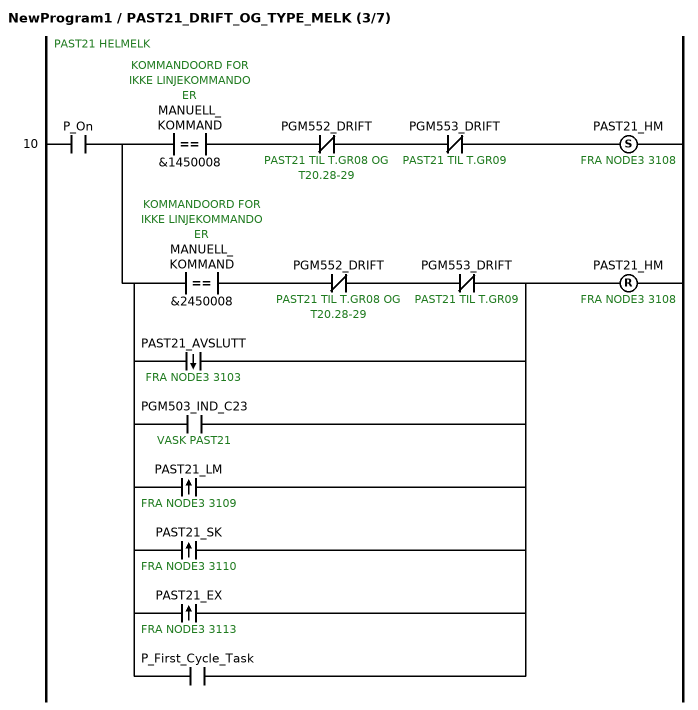
; [picture p1032: NewProgram1 / PAST21_DRIFT_OG_TYPE_MELK, rungs 10-10]
; rung 10: PAST21 HELMELK
LD P_On
OUT TR0
AND=L(301) MANUELL_KOMMAND &1450008  ; KOMMANDOORD FOR IKKE LINJEKOMMANDOER
ANDNOT PGM552_DRIFT  ; PAST21 TIL T.GR08 OG T20.28-29
ANDNOT PGM553_DRIFT  ; PAST21 TIL T.GR09
SET PAST21_HM  ; FRA NODE3 3108
LD TR0
LD=L(301) MANUELL_KOMMAND &2450008  ; KOMMANDOORD FOR IKKE LINJEKOMMANDOER
ANDNOT PGM552_DRIFT  ; PAST21 TIL T.GR08 OG T20.28-29
ANDNOT PGM553_DRIFT  ; PAST21 TIL T.GR09
%OR PAST21_AVSLUTT  ; FRA NODE3 3103
OR PGM503_IND_C23  ; VASK PAST21
@OR PAST21_LM  ; FRA NODE3 3109
@OR PAST21_SK  ; FRA NODE3 3110
@OR PAST21_EX  ; FRA NODE3 3113
OR P_First_Cycle_Task
ANDLD
RSET PAST21_HM  ; FRA NODE3 3108

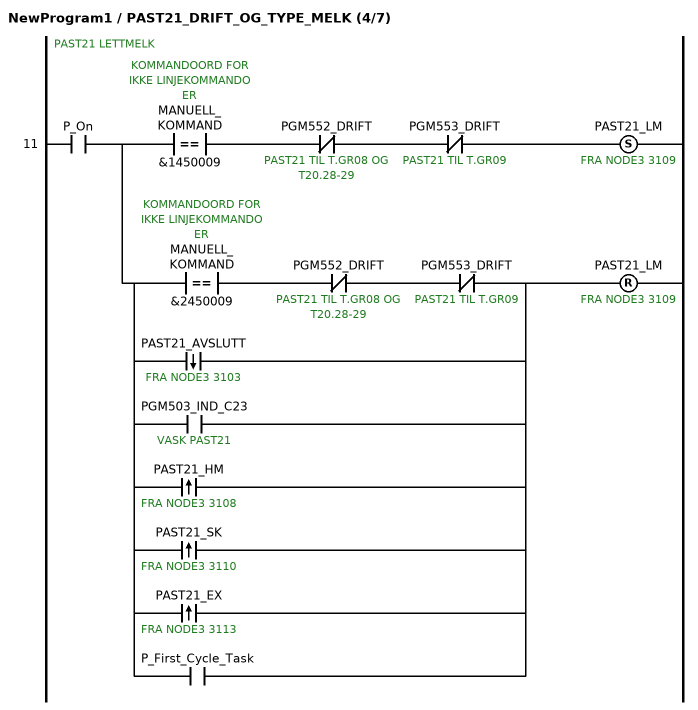
; rung 11: PAST21 LETTMELK
LD P_On
OUT TR0
AND=L(301) MANUELL_KOMMAND &1450009  ; KOMMANDOORD FOR IKKE LINJEKOMMANDOER
ANDNOT PGM552_DRIFT  ; PAST21 TIL T.GR08 OG T20.28-29
ANDNOT PGM553_DRIFT  ; PAST21 TIL T.GR09
SET PAST21_LM  ; FRA NODE3 3109
LD TR0
LD=L(301) MANUELL_KOMMAND &2450009  ; KOMMANDOORD FOR IKKE LINJEKOMMANDOER
ANDNOT PGM552_DRIFT  ; PAST21 TIL T.GR08 OG T20.28-29
ANDNOT PGM553_DRIFT  ; PAST21 TIL T.GR09
%OR PAST21_AVSLUTT  ; FRA NODE3 3103
OR PGM503_IND_C23  ; VASK PAST21
@OR PAST21_HM  ; FRA NODE3 3108
@OR PAST21_SK  ; FRA NODE3 3110
@OR PAST21_EX  ; FRA NODE3 3113
OR P_First_Cycle_Task
ANDLD
RSET PAST21_LM  ; FRA NODE3 3109

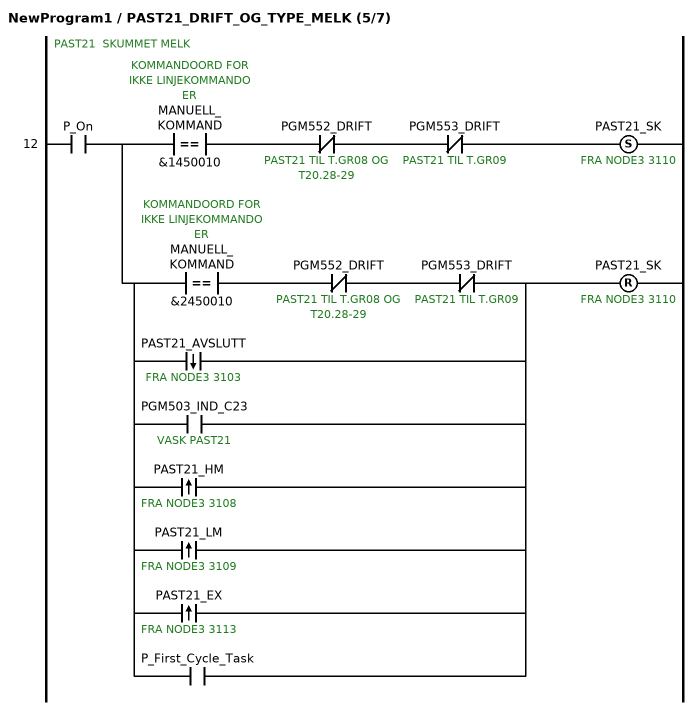
; rung 12: PAST21  SKUMMET MELK
LD P_On
OUT TR0
AND=L(301) MANUELL_KOMMAND &1450010  ; KOMMANDOORD FOR IKKE LINJEKOMMANDOER
ANDNOT PGM552_DRIFT  ; PAST21 TIL T.GR08 OG T20.28-29
ANDNOT PGM553_DRIFT  ; PAST21 TIL T.GR09
SET PAST21_SK  ; FRA NODE3 3110
LD TR0
LD=L(301) MANUELL_KOMMAND &2450010  ; KOMMANDOORD FOR IKKE LINJEKOMMANDOER
ANDNOT PGM552_DRIFT  ; PAST21 TIL T.GR08 OG T20.28-29
ANDNOT PGM553_DRIFT  ; PAST21 TIL T.GR09
%OR PAST21_AVSLUTT  ; FRA NODE3 3103
OR PGM503_IND_C23  ; VASK PAST21
@OR PAST21_HM  ; FRA NODE3 3108
@OR PAST21_LM  ; FRA NODE3 3109
@OR PAST21_EX  ; FRA NODE3 3113
OR P_First_Cycle_Task
ANDLD
RSET PAST21_SK  ; FRA NODE3 3110

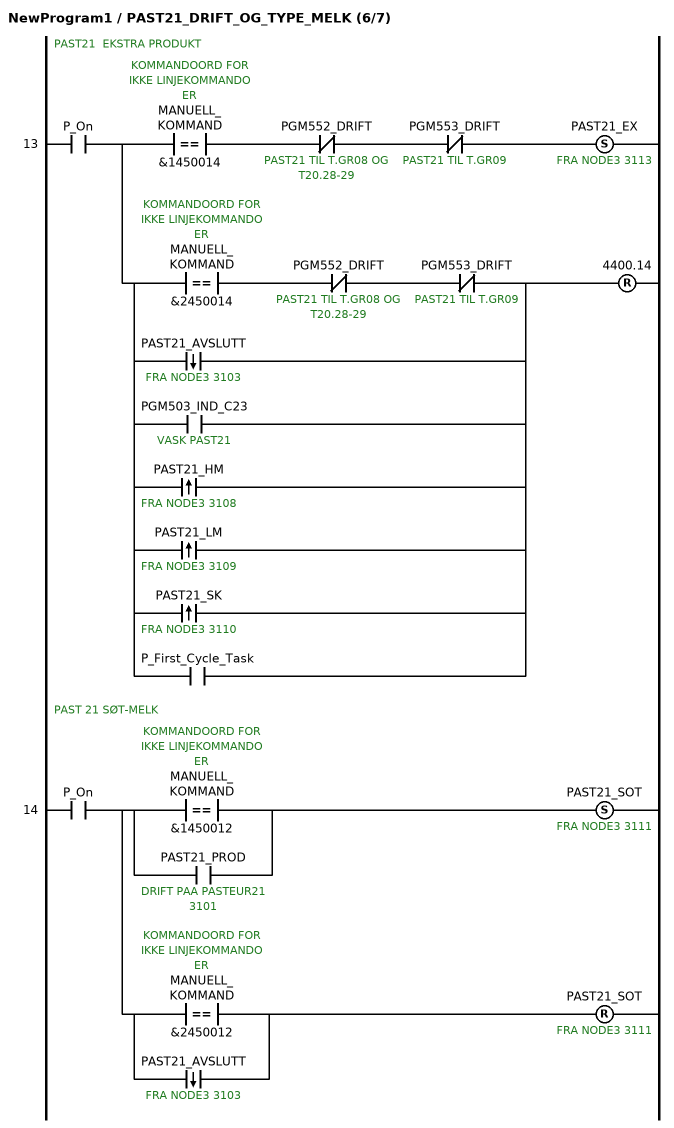
; rung 13: PAST21  EKSTRA PRODUKT
LD P_On
OUT TR0
AND=L(301) MANUELL_KOMMAND &1450014  ; KOMMANDOORD FOR IKKE LINJEKOMMANDOER
ANDNOT PGM552_DRIFT  ; PAST21 TIL T.GR08 OG T20.28-29
ANDNOT PGM553_DRIFT  ; PAST21 TIL T.GR09
SET PAST21_EX  ; FRA NODE3 3113
LD TR0
LD=L(301) MANUELL_KOMMAND &2450014  ; KOMMANDOORD FOR IKKE LINJEKOMMANDOER
ANDNOT PGM552_DRIFT  ; PAST21 TIL T.GR08 OG T20.28-29
ANDNOT PGM553_DRIFT  ; PAST21 TIL T.GR09
%OR PAST21_AVSLUTT  ; FRA NODE3 3103
OR PGM503_IND_C23  ; VASK PAST21
@OR PAST21_HM  ; FRA NODE3 3108
@OR PAST21_LM  ; FRA NODE3 3109
@OR PAST21_SK  ; FRA NODE3 3110
OR P_First_Cycle_Task
ANDLD
RSET 4400.14
; rung 14: PAST 21 SØT-MELK
LD P_On
OUT TR0
LD=L(301) MANUELL_KOMMAND &1450012  ; KOMMANDOORD FOR IKKE LINJEKOMMANDOER
OR PAST21_PROD  ; DRIFT PAA PASTEUR21 3101
ANDLD
SET PAST21_SOT  ; FRA NODE3 3111
LD TR0
LD=L(301) MANUELL_KOMMAND &2450012  ; KOMMANDOORD FOR IKKE LINJEKOMMANDOER
%OR PAST21_AVSLUTT  ; FRA NODE3 3103
ANDLD
RSET PAST21_SOT  ; FRA NODE3 3111

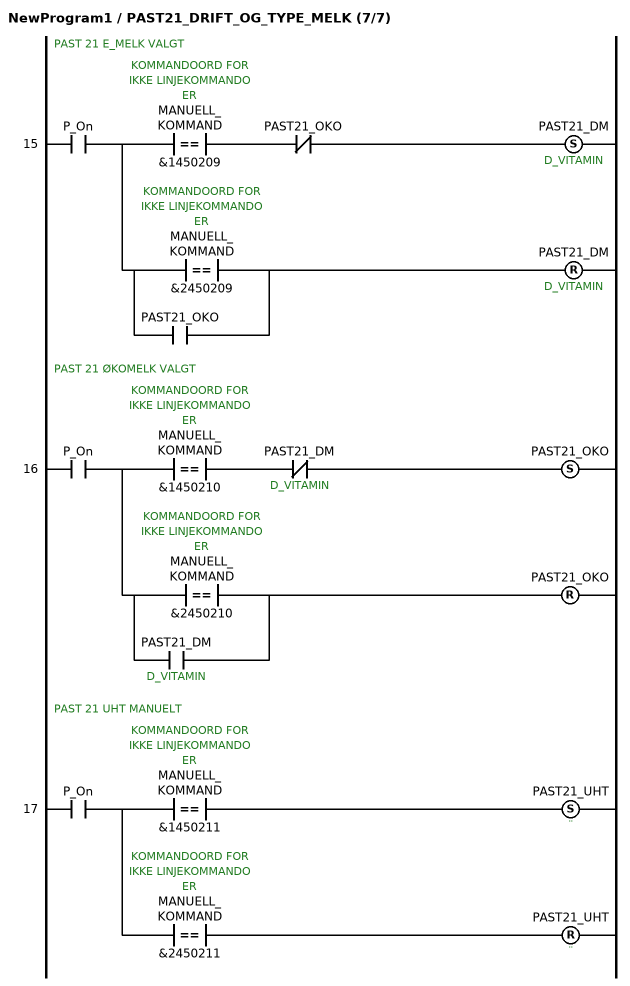
; rung 15: PAST 21 E_MELK VALGT
LD P_On
OUT TR0
AND=L(301) MANUELL_KOMMAND &1450209  ; KOMMANDOORD FOR IKKE LINJEKOMMANDOER
ANDNOT PAST21_OKO
SET PAST21_DM  ; D_VITAMIN
LD TR0
LD=L(301) MANUELL_KOMMAND &2450209  ; KOMMANDOORD FOR IKKE LINJEKOMMANDOER
OR PAST21_OKO
ANDLD
RSET PAST21_DM  ; D_VITAMIN
; rung 16: PAST 21 ØKOMELK VALGT
LD P_On
OUT TR0
AND=L(301) MANUELL_KOMMAND &1450210  ; KOMMANDOORD FOR IKKE LINJEKOMMANDOER
ANDNOT PAST21_DM  ; D_VITAMIN
SET PAST21_OKO
LD TR0
LD=L(301) MANUELL_KOMMAND &2450210  ; KOMMANDOORD FOR IKKE LINJEKOMMANDOER
OR PAST21_DM  ; D_VITAMIN
ANDLD
RSET PAST21_OKO
; rung 17: PAST 21 UHT MANUELT
LD P_On
OUT TR0
AND=L(301) MANUELL_KOMMAND &1450211  ; KOMMANDOORD FOR IKKE LINJEKOMMANDOER
SET PAST21_UHT  ; ¨
LD TR0
AND=L(301) MANUELL_KOMMAND &2450211  ; KOMMANDOORD FOR IKKE LINJEKOMMANDOER
RSET PAST21_UHT  ; ¨
; rung 18: Ingen_kommentar_funnet

### Section PAST21_STATUSKONTROLL

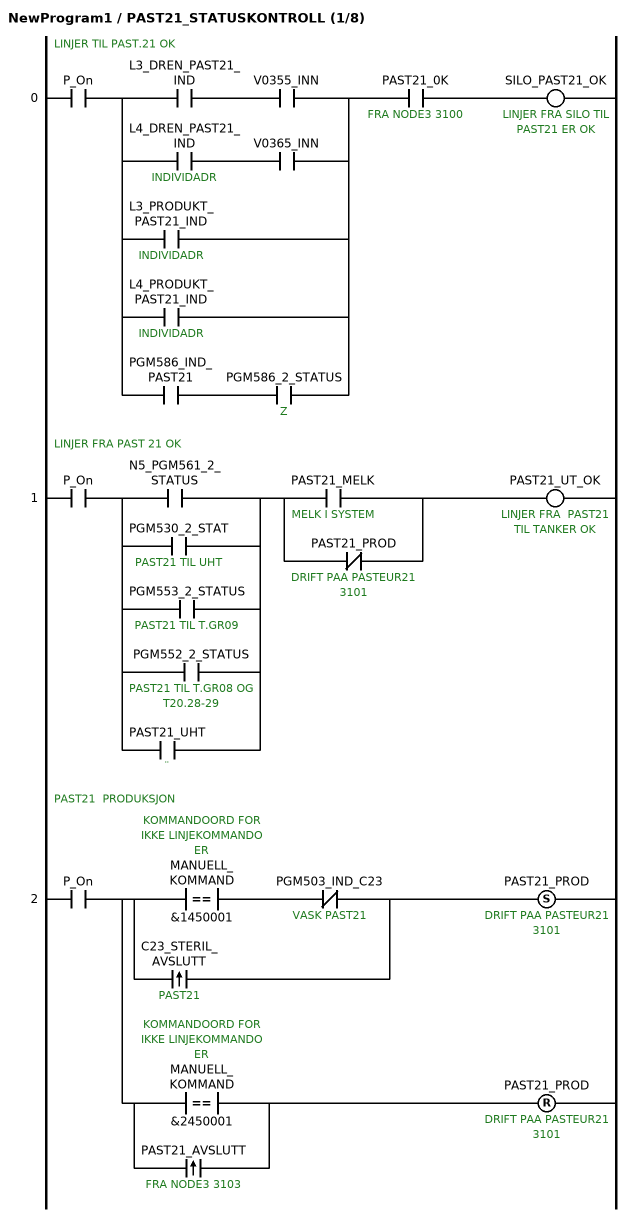
; rung 0: LINJER TIL PAST.21 OK
LD P_On
LD L3_DREN_PAST21_IND
AND V0355_INN
LD L4_DREN_PAST21_IND  ; INDIVIDADR
AND V0365_INN
ORLD
OR L3_PRODUKT_PAST21_IND  ; INDIVIDADR
OR L4_PRODUKT_PAST21_IND  ; INDIVIDADR
LD PGM586_IND_PAST21
AND PGM586_2_STATUS  ; Z
ORLD
ANDLD
AND PAST21_0K  ; FRA NODE3 3100
OUT SILO_PAST21_OK  ; LINJER FRA SILO TIL  PAST21 ER OK
; rung 1: LINJER FRA PAST 21 OK
LD P_On
LD N5_PGM561_2_STATUS
OR PGM530_2_STAT  ; PAST21 TIL UHT
OR PGM553_2_STATUS  ; PAST21 TIL T.GR09
OR PGM552_2_STATUS  ; PAST21 TIL T.GR08 OG T20.28-29
OR PAST21_UHT  ; ¨
ANDLD
LD PAST21_MELK  ; MELK I SYSTEM
ORNOT PAST21_PROD  ; DRIFT PAA PASTEUR21 3101
ANDLD
OUT PAST21_UT_OK  ; LINJER FRA  PAST21 TIL TANKER OK
; rung 2: PAST21  PRODUKSJON
LD P_On
OUT TR0
LD=L(301) MANUELL_KOMMAND &1450001  ; KOMMANDOORD FOR IKKE LINJEKOMMANDOER
ANDNOT PGM503_IND_C23  ; VASK PAST21
@OR C23_STERIL_AVSLUTT  ; PAST21
ANDLD
SET PAST21_PROD  ; DRIFT PAA PASTEUR21 3101
LD TR0
LD=L(301) MANUELL_KOMMAND &2450001  ; KOMMANDOORD FOR IKKE LINJEKOMMANDOER
@OR PAST21_AVSLUTT  ; FRA NODE3 3103
ANDLD
RSET PAST21_PROD  ; DRIFT PAA PASTEUR21 3101

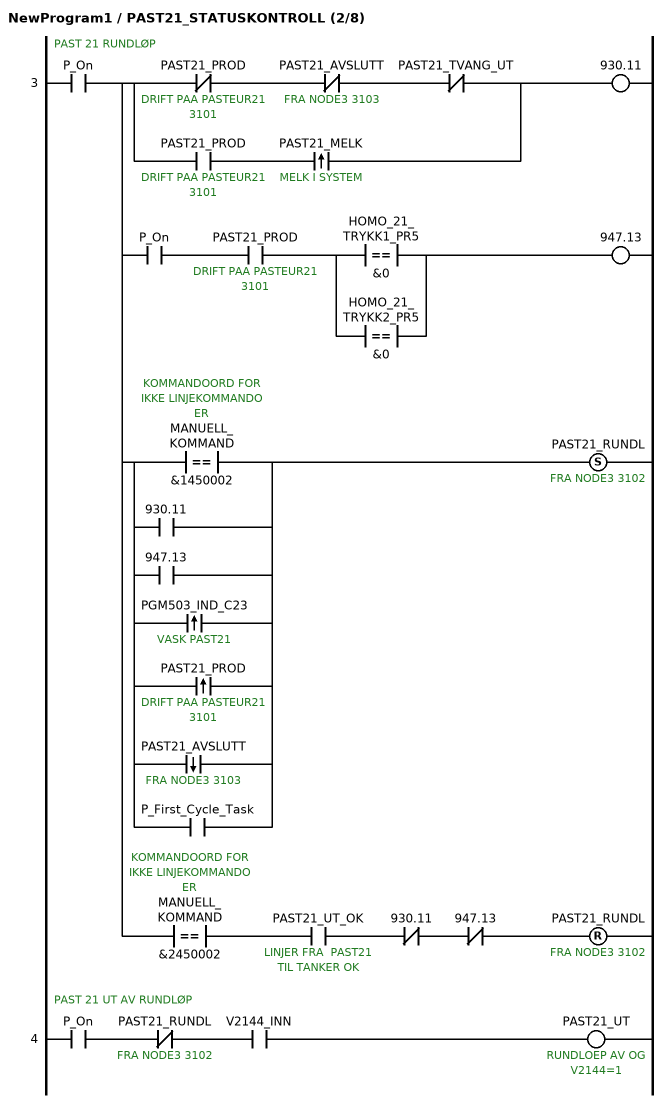
; rung 3: PAST 21 RUNDLØP
LD P_On
OUT TR0
LDNOT PAST21_PROD  ; DRIFT PAA PASTEUR21 3101
ANDNOT PAST21_AVSLUTT  ; FRA NODE3 3103
ANDNOT PAST21_TVANG_UT
LD PAST21_PROD  ; DRIFT PAA PASTEUR21 3101
@AND PAST21_MELK  ; MELK I SYSTEM
ORLD
ANDLD
OUT 930.11
LD TR0
AND P_On
AND PAST21_PROD  ; DRIFT PAA PASTEUR21 3101
LD=L(301) HOMO_21_TRYKK1_PR5 &0
OR=L(301) HOMO_21_TRYKK2_PR5 &0
ANDLD
OUT 947.13
LD TR0
LD=L(301) MANUELL_KOMMAND &1450002  ; KOMMANDOORD FOR IKKE LINJEKOMMANDOER
OR 930.11
OR 947.13
@OR PGM503_IND_C23  ; VASK PAST21
@OR PAST21_PROD  ; DRIFT PAA PASTEUR21 3101
%OR PAST21_AVSLUTT  ; FRA NODE3 3103
OR P_First_Cycle_Task
ANDLD
SET PAST21_RUNDL  ; FRA NODE3 3102
LD TR0
AND=L(301) MANUELL_KOMMAND &2450002  ; KOMMANDOORD FOR IKKE LINJEKOMMANDOER
AND PAST21_UT_OK  ; LINJER FRA  PAST21 TIL TANKER OK
ANDNOT 930.11
ANDNOT 947.13
RSET PAST21_RUNDL  ; FRA NODE3 3102
; rung 4: PAST 21 UT AV RUNDLØP
LD P_On
ANDNOT PAST21_RUNDL  ; FRA NODE3 3102
AND V2144_INN
OUT PAST21_UT  ; RUNDLOEP AV OG V2144=1

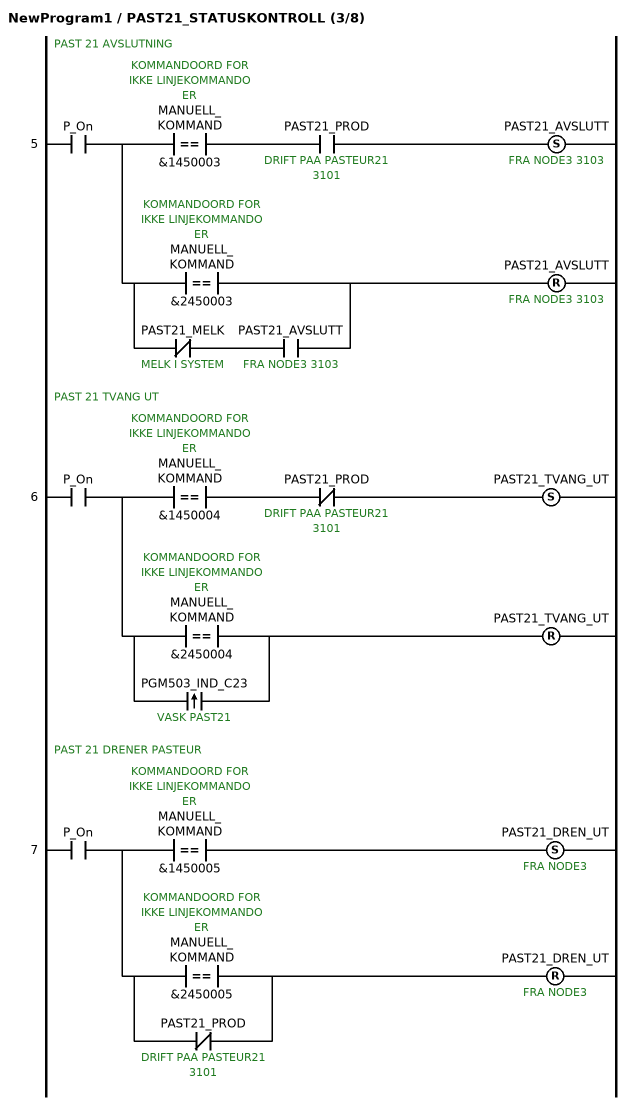
; rung 5: PAST 21 AVSLUTNING
LD P_On
OUT TR0
AND=L(301) MANUELL_KOMMAND &1450003  ; KOMMANDOORD FOR IKKE LINJEKOMMANDOER
AND PAST21_PROD  ; DRIFT PAA PASTEUR21 3101
SET PAST21_AVSLUTT  ; FRA NODE3 3103
LD TR0
LD=L(301) MANUELL_KOMMAND &2450003  ; KOMMANDOORD FOR IKKE LINJEKOMMANDOER
LDNOT PAST21_MELK  ; MELK I SYSTEM
AND PAST21_AVSLUTT  ; FRA NODE3 3103
ORLD
ANDLD
RSET PAST21_AVSLUTT  ; FRA NODE3 3103
; rung 6: PAST 21 TVANG UT
LD P_On
OUT TR0
AND=L(301) MANUELL_KOMMAND &1450004  ; KOMMANDOORD FOR IKKE LINJEKOMMANDOER
ANDNOT PAST21_PROD  ; DRIFT PAA PASTEUR21 3101
SET PAST21_TVANG_UT
LD TR0
LD=L(301) MANUELL_KOMMAND &2450004  ; KOMMANDOORD FOR IKKE LINJEKOMMANDOER
@OR PGM503_IND_C23  ; VASK PAST21
ANDLD
RSET PAST21_TVANG_UT
; rung 7: PAST 21 DRENER PASTEUR
LD P_On
OUT TR0
AND=L(301) MANUELL_KOMMAND &1450005  ; KOMMANDOORD FOR IKKE LINJEKOMMANDOER
SET PAST21_DREN_UT  ; FRA NODE3
LD TR0
LD=L(301) MANUELL_KOMMAND &2450005  ; KOMMANDOORD FOR IKKE LINJEKOMMANDOER
ORNOT PAST21_PROD  ; DRIFT PAA PASTEUR21 3101
ANDLD
RSET PAST21_DREN_UT  ; FRA NODE3

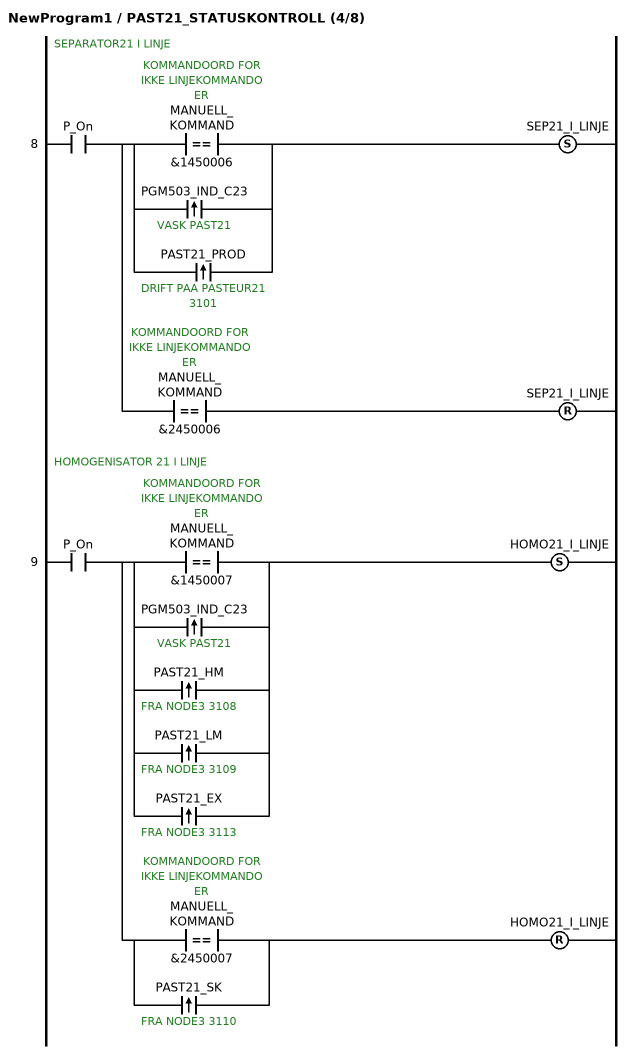
; rung 8: SEPARATOR21 I LINJE
LD P_On
OUT TR0
LD=L(301) MANUELL_KOMMAND &1450006  ; KOMMANDOORD FOR IKKE LINJEKOMMANDOER
@OR PGM503_IND_C23  ; VASK PAST21
@OR PAST21_PROD  ; DRIFT PAA PASTEUR21 3101
ANDLD
SET SEP21_I_LINJE
LD TR0
AND=L(301) MANUELL_KOMMAND &2450006  ; KOMMANDOORD FOR IKKE LINJEKOMMANDOER
RSET SEP21_I_LINJE
; rung 9: HOMOGENISATOR 21 I LINJE
LD P_On
OUT TR0
LD=L(301) MANUELL_KOMMAND &1450007  ; KOMMANDOORD FOR IKKE LINJEKOMMANDOER
@OR PGM503_IND_C23  ; VASK PAST21
@OR PAST21_HM  ; FRA NODE3 3108
@OR PAST21_LM  ; FRA NODE3 3109
@OR PAST21_EX  ; FRA NODE3 3113
ANDLD
SET HOMO21_I_LINJE
LD TR0
LD=L(301) MANUELL_KOMMAND &2450007  ; KOMMANDOORD FOR IKKE LINJEKOMMANDOER
@OR PAST21_SK  ; FRA NODE3 3110
ANDLD
RSET HOMO21_I_LINJE

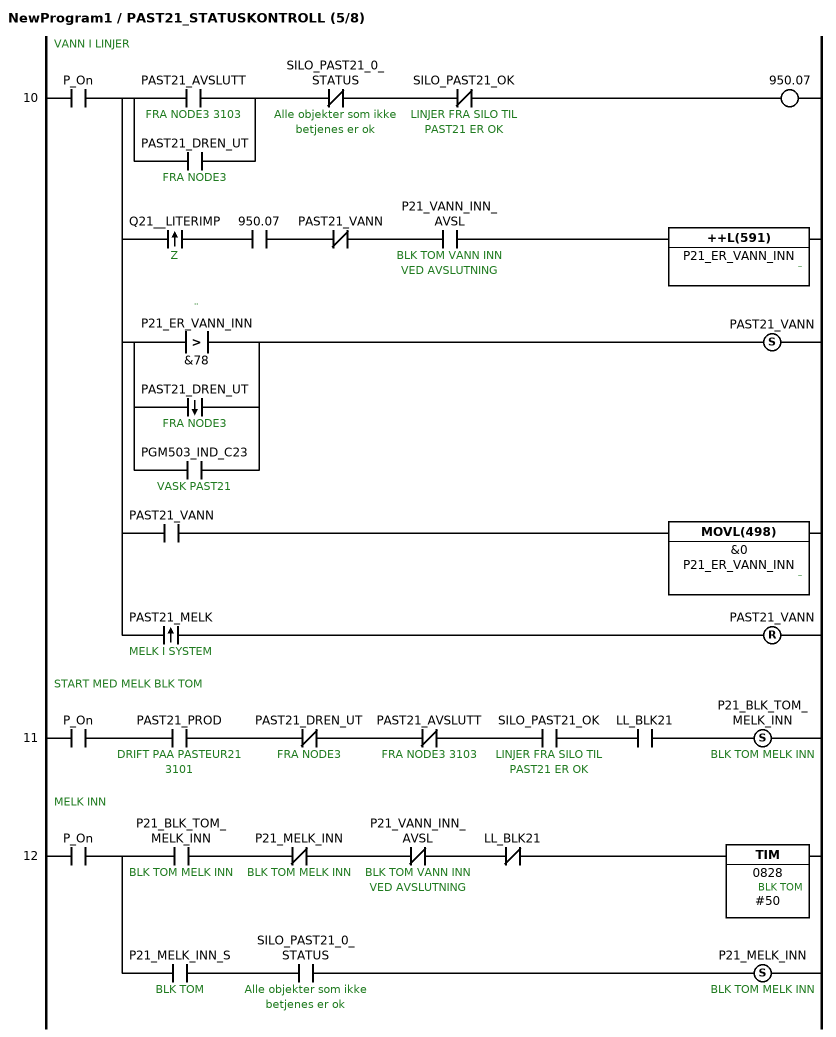
; rung 10: VANN I LINJER
LD P_On
OUT TR0
LD PAST21_AVSLUTT  ; FRA NODE3 3103
OR PAST21_DREN_UT  ; FRA NODE3
ANDLD
ANDNOT SILO_PAST21_0_STATUS  ; Alle objekter som ikke betjenes er ok
ANDNOT SILO_PAST21_OK  ; LINJER FRA SILO TIL  PAST21 ER OK
OUT 950.07
LD TR0
@AND Q21__LITERIMP  ; Z
AND 950.07
ANDNOT PAST21_VANN
AND P21_VANN_INN_AVSL  ; BLK TOM VANN INN VED AVSLUTNING
++L(591) P21_ER_VANN_INN  ; ¨
LD TR0
LD>L(321) P21_ER_VANN_INN &78  ; ¨
%OR PAST21_DREN_UT  ; FRA NODE3
OR PGM503_IND_C23  ; VASK PAST21
ANDLD
SET PAST21_VANN
LD TR0
AND PAST21_VANN
MOVL(498) &0 P21_ER_VANN_INN  ; ¨
LD TR0
@AND PAST21_MELK  ; MELK I SYSTEM
RSET PAST21_VANN
; rung 11: START MED MELK BLK TOM
LD P_On
AND PAST21_PROD  ; DRIFT PAA PASTEUR21 3101
ANDNOT PAST21_DREN_UT  ; FRA NODE3
ANDNOT PAST21_AVSLUTT  ; FRA NODE3 3103
AND SILO_PAST21_OK  ; LINJER FRA SILO TIL  PAST21 ER OK
AND LL_BLK21
SET P21_BLK_TOM_MELK_INN  ; BLK TOM MELK INN
; rung 12: MELK INN
LD P_On
OUT TR0
AND P21_BLK_TOM_MELK_INN  ; BLK TOM MELK INN
ANDNOT P21_MELK_INN  ; BLK TOM MELK INN
ANDNOT P21_VANN_INN_AVSL  ; BLK TOM VANN INN VED AVSLUTNING
ANDNOT LL_BLK21
TIM 0828 #50  ; BLK TOM
LD TR0
AND P21_MELK_INN_S  ; BLK TOM
AND SILO_PAST21_0_STATUS  ; Alle objekter som ikke betjenes er ok
SET P21_MELK_INN  ; BLK TOM MELK INN

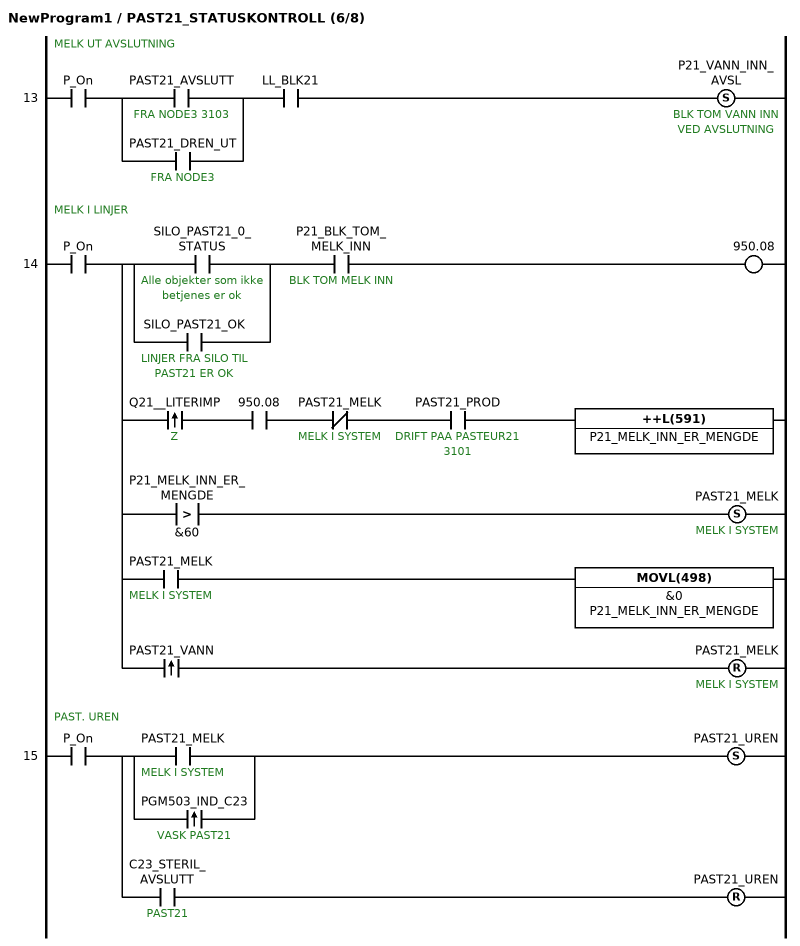
; rung 13: MELK UT AVSLUTNING
LD P_On
LD PAST21_AVSLUTT  ; FRA NODE3 3103
OR PAST21_DREN_UT  ; FRA NODE3
ANDLD
AND LL_BLK21
SET P21_VANN_INN_AVSL  ; BLK TOM VANN INN VED AVSLUTNING
; rung 14: MELK I LINJER
LD P_On
OUT TR0
LD SILO_PAST21_0_STATUS  ; Alle objekter som ikke betjenes er ok
OR SILO_PAST21_OK  ; LINJER FRA SILO TIL  PAST21 ER OK
ANDLD
AND P21_BLK_TOM_MELK_INN  ; BLK TOM MELK INN
OUT 950.08
LD TR0
@AND Q21__LITERIMP  ; Z
AND 950.08
ANDNOT PAST21_MELK  ; MELK I SYSTEM
AND PAST21_PROD  ; DRIFT PAA PASTEUR21 3101
++L(591) P21_MELK_INN_ER_MENGDE
LD TR0
AND>L(321) P21_MELK_INN_ER_MENGDE &60
SET PAST21_MELK  ; MELK I SYSTEM
LD TR0
AND PAST21_MELK  ; MELK I SYSTEM
MOVL(498) &0 P21_MELK_INN_ER_MENGDE
LD TR0
@AND PAST21_VANN
RSET PAST21_MELK  ; MELK I SYSTEM
; rung 15: PAST. UREN
LD P_On
OUT TR0
LD PAST21_MELK  ; MELK I SYSTEM
@OR PGM503_IND_C23  ; VASK PAST21
ANDLD
SET PAST21_UREN
LD TR0
AND C23_STERIL_AVSLUTT  ; PAST21
RSET PAST21_UREN

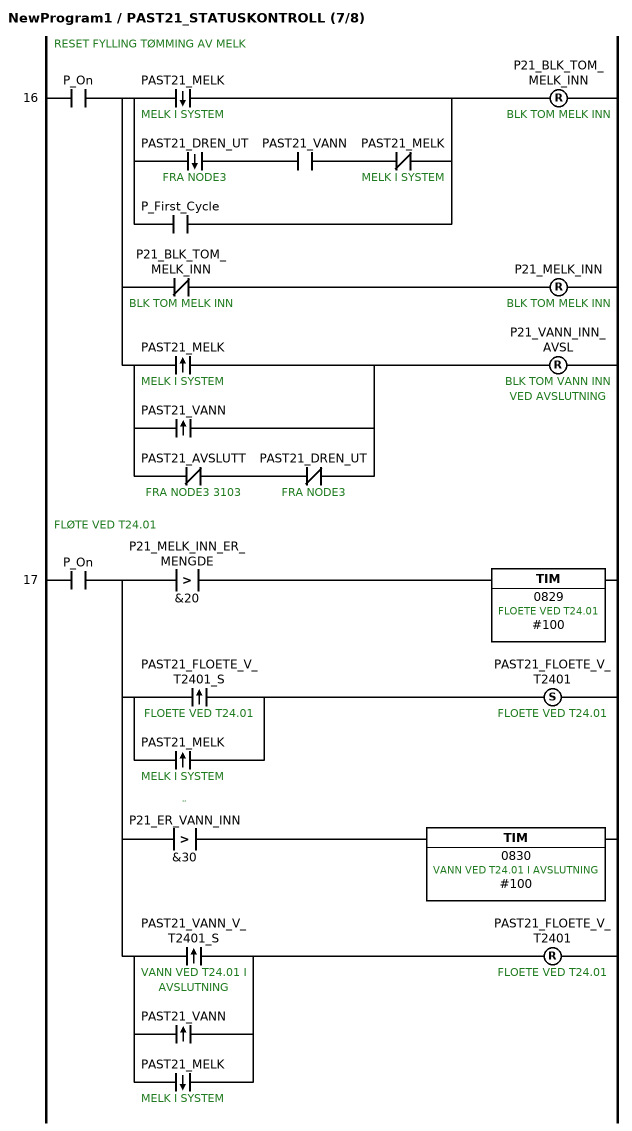
; rung 16: RESET FYLLING TØMMING AV MELK
LD P_On
OUT TR0
%LD PAST21_MELK  ; MELK I SYSTEM
%LD PAST21_DREN_UT  ; FRA NODE3
AND PAST21_VANN
ANDNOT PAST21_MELK  ; MELK I SYSTEM
ORLD
OR P_First_Cycle
ANDLD
RSET P21_BLK_TOM_MELK_INN  ; BLK TOM MELK INN
LD TR0
ANDNOT P21_BLK_TOM_MELK_INN  ; BLK TOM MELK INN
RSET P21_MELK_INN  ; BLK TOM MELK INN
LD TR0
@LD PAST21_MELK  ; MELK I SYSTEM
@OR PAST21_VANN
LDNOT PAST21_AVSLUTT  ; FRA NODE3 3103
ANDNOT PAST21_DREN_UT  ; FRA NODE3
ORLD
ANDLD
RSET P21_VANN_INN_AVSL  ; BLK TOM VANN INN VED AVSLUTNING
; rung 17: FLØTE VED T24.01
LD P_On
OUT TR0
AND>L(321) P21_MELK_INN_ER_MENGDE &20
TIM 0829 #100  ; FLOETE VED T24.01
LD TR0
@LD PAST21_FLOETE_V_T2401_S  ; FLOETE VED T24.01
@OR PAST21_MELK  ; MELK I SYSTEM
ANDLD
SET PAST21_FLOETE_V_T2401  ; FLOETE VED T24.01
LD TR0
AND>L(321) P21_ER_VANN_INN &30  ; ¨
TIM 0830 #100  ; VANN VED T24.01 I AVSLUTNING
LD TR0
@LD PAST21_VANN_V_T2401_S  ; VANN VED T24.01 I AVSLUTNING
@OR PAST21_VANN
%OR PAST21_MELK  ; MELK I SYSTEM
ANDLD
RSET PAST21_FLOETE_V_T2401  ; FLOETE VED T24.01

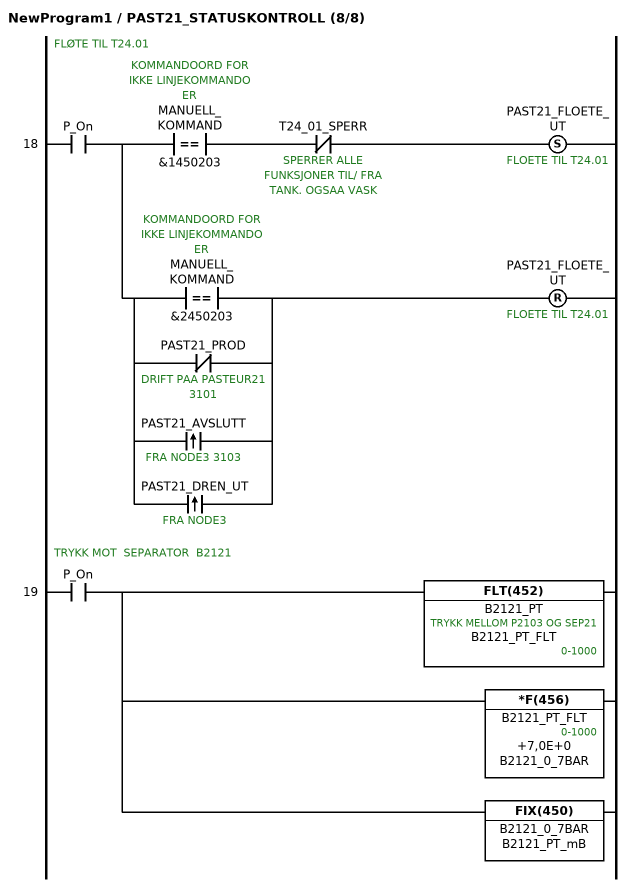
; rung 18: FLØTE TIL T24.01
LD P_On
OUT TR0
AND=L(301) MANUELL_KOMMAND &1450203  ; KOMMANDOORD FOR IKKE LINJEKOMMANDOER
ANDNOT T24_01_SPERR  ; SPERRER ALLE FUNKSJONER TIL/ FRA TANK. OGSAA VASK
SET PAST21_FLOETE_UT  ; FLOETE TIL T24.01
LD TR0
LD=L(301) MANUELL_KOMMAND &2450203  ; KOMMANDOORD FOR IKKE LINJEKOMMANDOER
ORNOT PAST21_PROD  ; DRIFT PAA PASTEUR21 3101
@OR PAST21_AVSLUTT  ; FRA NODE3 3103
@OR PAST21_DREN_UT  ; FRA NODE3
ANDLD
RSET PAST21_FLOETE_UT  ; FLOETE TIL T24.01
; rung 19: TRYKK MOT  SEPARATOR  B2121
LD P_On
FLT(452) B2121_PT B2121_PT_FLT  ; TRYKK MELLOM P2103 OG SEP21, 0-1000
*F(456) B2121_PT_FLT +7,0E+0 B2121_0_7BAR  ; 0-1000
FIX(450) B2121_0_7BAR B2121_PT_mB
; rung 20: Ingen_kommentar_funnet

### Section PAST21_OMSLAGSKONTROLL
; PÅL

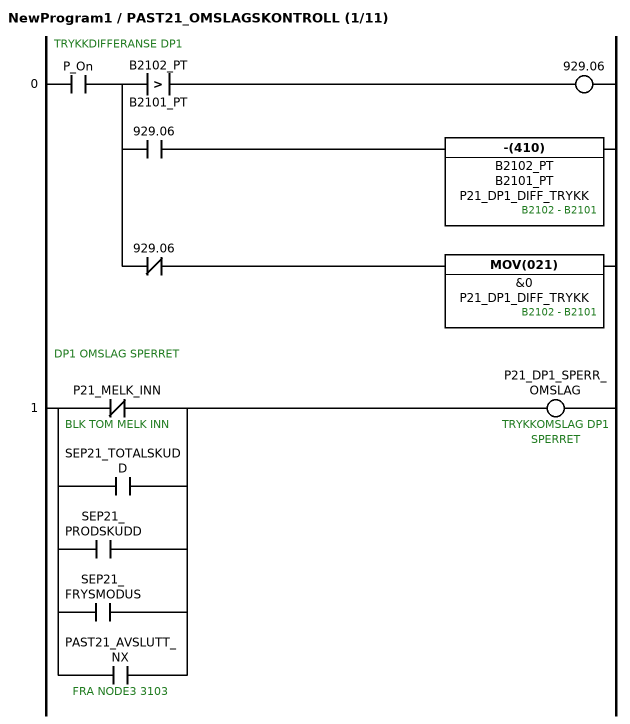
; rung 0: TRYKKDIFFERANSE DP1
LD P_On
OUT TR0
AND>(320) B2102_PT B2101_PT
OUT 929.06
LD TR0
AND 929.06
-(410) B2102_PT B2101_PT P21_DP1_DIFF_TRYKK  ; B2102 - B2101
LD TR0
ANDNOT 929.06
MOV(021) &0 P21_DP1_DIFF_TRYKK  ; B2102 - B2101
; rung 1: DP1 OMSLAG SPERRET
LDNOT P21_MELK_INN  ; BLK TOM MELK INN
OR SEP21_TOTALSKUDD
OR SEP21_PRODSKUDD
OR SEP21_FRYSMODUS
OR PAST21_AVSLUTT_NX  ; FRA NODE3 3103
OUT P21_DP1_SPERR_OMSLAG  ; TRYKKOMSLAG DP1 SPERRET

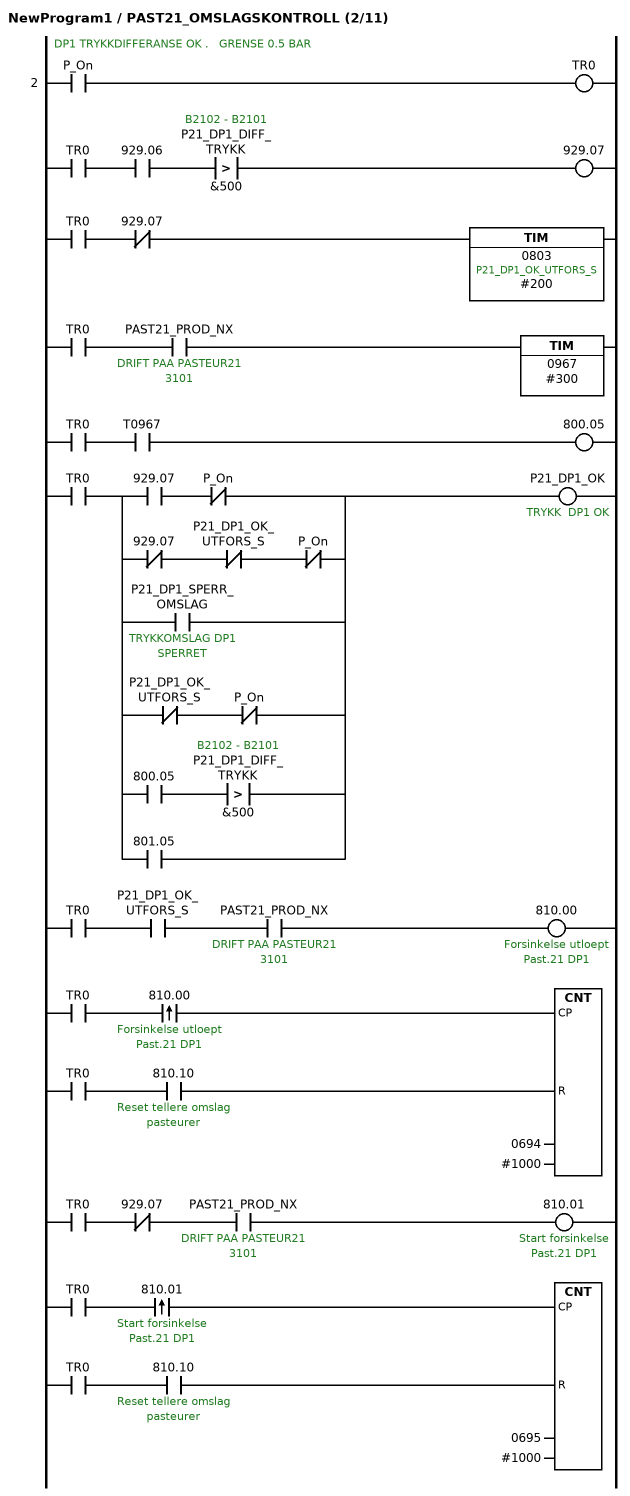
; rung 2: DP1 TRYKKDIFFERANSE OK .   GRENSE 0.5 BAR
LD P_On
OUT TR0
AND 929.06
AND>(320) P21_DP1_DIFF_TRYKK &500  ; B2102 - B2101
OUT 929.07
LD TR0
ANDNOT 929.07
TIM 0803 #200  ; P21_DP1_OK_UTFORS_S
LD TR0
AND PAST21_PROD_NX  ; DRIFT PAA PASTEUR21 3101
TIM 0967 #300
LD TR0
AND T0967
OUT 800.05
LD TR0
LD 929.07
ANDNOT P_On
LDNOT 929.07
ANDNOT P21_DP1_OK_UTFORS_S
ANDNOT P_On
ORLD
OR P21_DP1_SPERR_OMSLAG  ; TRYKKOMSLAG DP1 SPERRET
LDNOT P21_DP1_OK_UTFORS_S
ANDNOT P_On
ORLD
LD 800.05
AND>(320) P21_DP1_DIFF_TRYKK &500  ; B2102 - B2101
ORLD
OR 801.05
ANDLD
OUT P21_DP1_OK  ; TRYKK  DP1 OK
LD TR0
AND P21_DP1_OK_UTFORS_S
AND PAST21_PROD_NX  ; DRIFT PAA PASTEUR21 3101
OUT 810.00  ; Forsinkelse utloept Past.21 DP1
LD TR0
@AND 810.00  ; Forsinkelse utloept Past.21 DP1
LD TR0
AND 810.10  ; Reset tellere omslag pasteurer
CNT 0694 #1000
LD TR0
ANDNOT 929.07
AND PAST21_PROD_NX  ; DRIFT PAA PASTEUR21 3101
OUT 810.01  ; Start forsinkelse Past.21 DP1
LD TR0
@AND 810.01  ; Start forsinkelse Past.21 DP1
LD TR0
AND 810.10  ; Reset tellere omslag pasteurer
CNT 0695 #1000

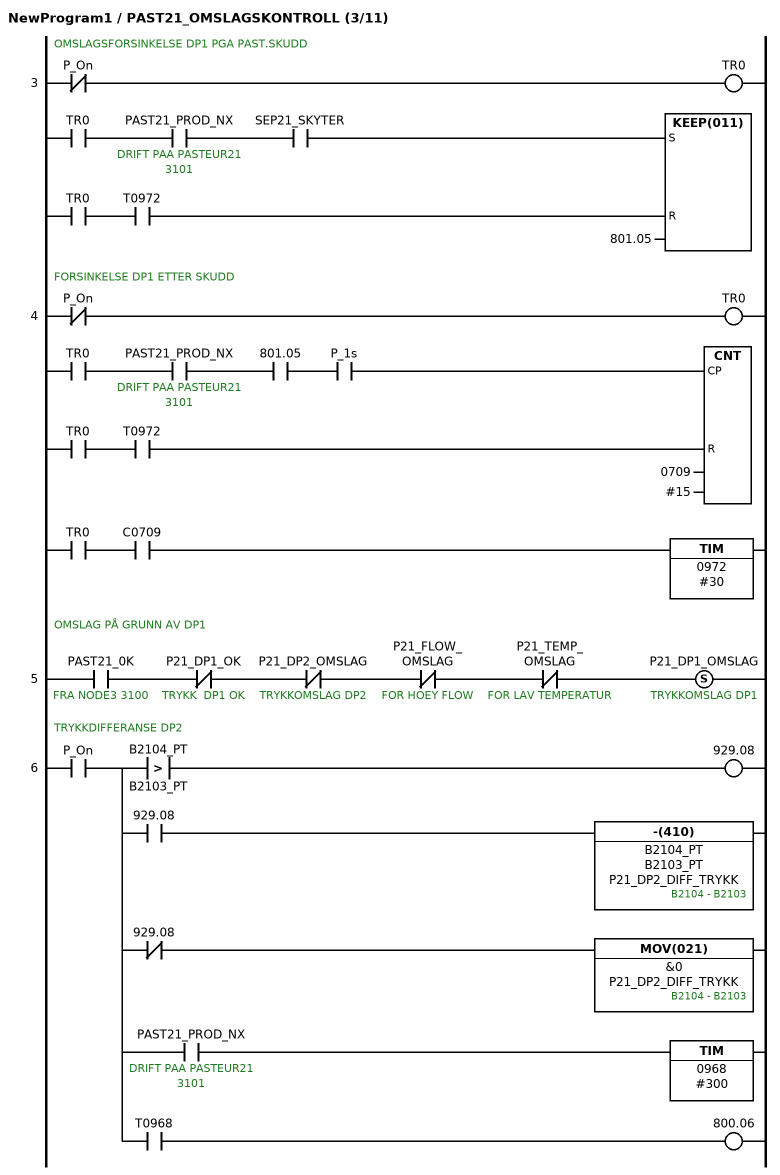
; rung 3: OMSLAGSFORSINKELSE DP1 PGA PAST.SKUDD
LDNOT P_On
OUT TR0
AND PAST21_PROD_NX  ; DRIFT PAA PASTEUR21 3101
AND SEP21_SKYTER
LD TR0
AND T0972
KEEP(011) 801.05
; rung 4: FORSINKELSE DP1 ETTER SKUDD
LDNOT P_On
OUT TR0
AND PAST21_PROD_NX  ; DRIFT PAA PASTEUR21 3101
AND 801.05
AND P_1s
LD TR0
AND T0972
CNT 0709 #15
LD TR0
AND C0709
TIM 0972 #30
; rung 5: OMSLAG PÅ GRUNN AV DP1
LD PAST21_0K  ; FRA NODE3 3100
ANDNOT P21_DP1_OK  ; TRYKK  DP1 OK
ANDNOT P21_DP2_OMSLAG  ; TRYKKOMSLAG DP2
ANDNOT P21_FLOW_OMSLAG  ; FOR HOEY FLOW
ANDNOT P21_TEMP_OMSLAG  ; FOR LAV TEMPERATUR
SET P21_DP1_OMSLAG  ; TRYKKOMSLAG DP1
; rung 6: TRYKKDIFFERANSE DP2
LD P_On
OUT TR0
AND>(320) B2104_PT B2103_PT
OUT 929.08
LD TR0
AND 929.08
-(410) B2104_PT B2103_PT P21_DP2_DIFF_TRYKK  ; B2104 - B2103
LD TR0
ANDNOT 929.08
MOV(021) &0 P21_DP2_DIFF_TRYKK  ; B2104 - B2103
LD TR0
AND PAST21_PROD_NX  ; DRIFT PAA PASTEUR21 3101
TIM 0968 #300
LD TR0
AND T0968
OUT 800.06

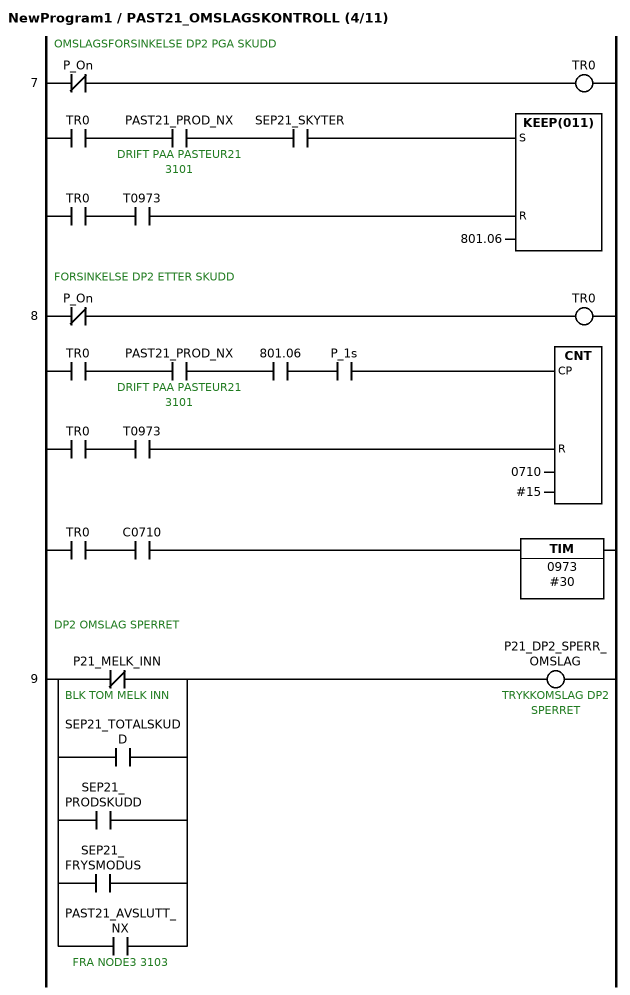
; rung 7: OMSLAGSFORSINKELSE DP2 PGA SKUDD
LDNOT P_On
OUT TR0
AND PAST21_PROD_NX  ; DRIFT PAA PASTEUR21 3101
AND SEP21_SKYTER
LD TR0
AND T0973
KEEP(011) 801.06
; rung 8: FORSINKELSE DP2 ETTER SKUDD
LDNOT P_On
OUT TR0
AND PAST21_PROD_NX  ; DRIFT PAA PASTEUR21 3101
AND 801.06
AND P_1s
LD TR0
AND T0973
CNT 0710 #15
LD TR0
AND C0710
TIM 0973 #30
; rung 9: DP2 OMSLAG SPERRET
LDNOT P21_MELK_INN  ; BLK TOM MELK INN
OR SEP21_TOTALSKUDD
OR SEP21_PRODSKUDD
OR SEP21_FRYSMODUS
OR PAST21_AVSLUTT_NX  ; FRA NODE3 3103
OUT P21_DP2_SPERR_OMSLAG  ; TRYKKOMSLAG DP2 SPERRET

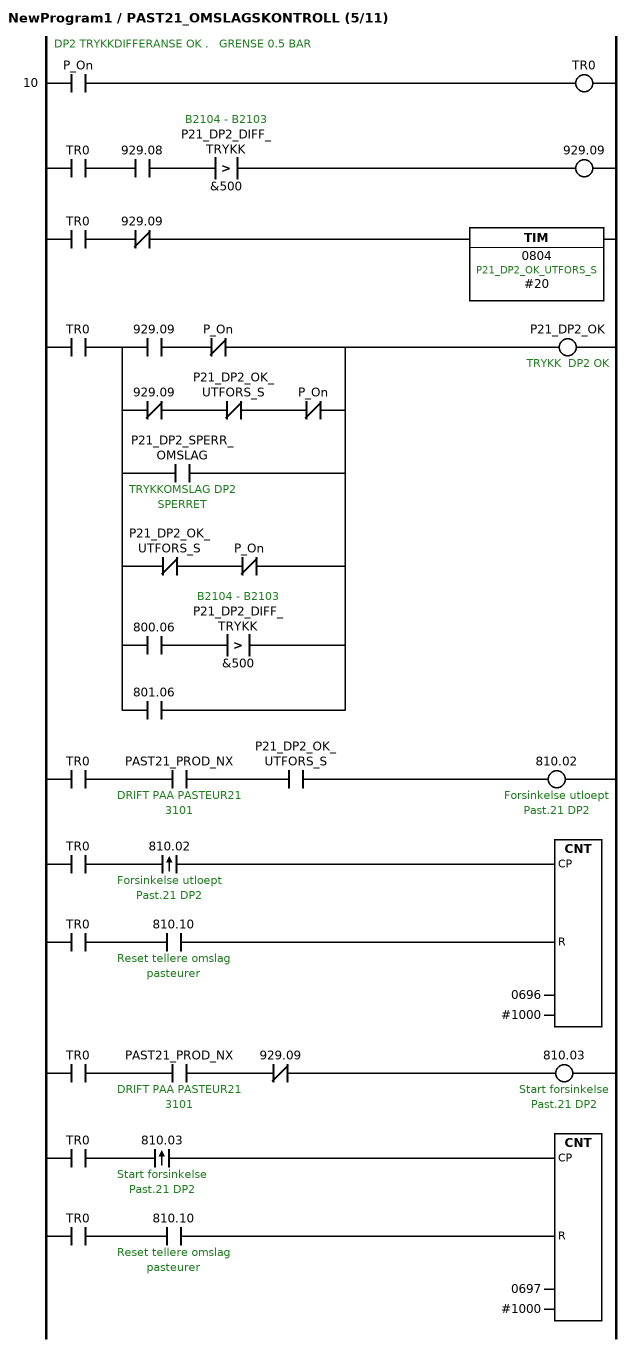
; rung 10: DP2 TRYKKDIFFERANSE OK .   GRENSE 0.5 BAR
LD P_On
OUT TR0
AND 929.08
AND>(320) P21_DP2_DIFF_TRYKK &500  ; B2104 - B2103
OUT 929.09
LD TR0
ANDNOT 929.09
TIM 0804 #20  ; P21_DP2_OK_UTFORS_S
LD TR0
LD 929.09
ANDNOT P_On
LDNOT 929.09
ANDNOT P21_DP2_OK_UTFORS_S
ANDNOT P_On
ORLD
OR P21_DP2_SPERR_OMSLAG  ; TRYKKOMSLAG DP2 SPERRET
LDNOT P21_DP2_OK_UTFORS_S
ANDNOT P_On
ORLD
LD 800.06
AND>(320) P21_DP2_DIFF_TRYKK &500  ; B2104 - B2103
ORLD
OR 801.06
ANDLD
OUT P21_DP2_OK  ; TRYKK  DP2 OK
LD TR0
AND PAST21_PROD_NX  ; DRIFT PAA PASTEUR21 3101
AND P21_DP2_OK_UTFORS_S
OUT 810.02  ; Forsinkelse utloept Past.21 DP2
LD TR0
@AND 810.02  ; Forsinkelse utloept Past.21 DP2
LD TR0
AND 810.10  ; Reset tellere omslag pasteurer
CNT 0696 #1000
LD TR0
AND PAST21_PROD_NX  ; DRIFT PAA PASTEUR21 3101
ANDNOT 929.09
OUT 810.03  ; Start forsinkelse Past.21 DP2
LD TR0
@AND 810.03  ; Start forsinkelse Past.21 DP2
LD TR0
AND 810.10  ; Reset tellere omslag pasteurer
CNT 0697 #1000

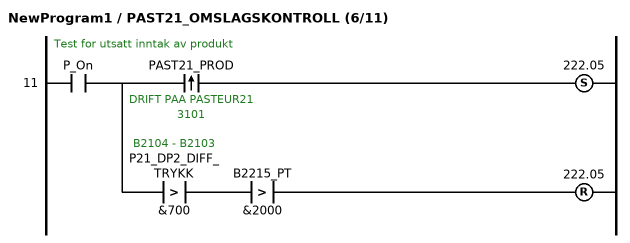
; rung 11: Test for utsatt inntak av produkt
LD P_On
OUT TR0
@AND PAST21_PROD  ; DRIFT PAA PASTEUR21 3101
SET 222.05
LD TR0
AND>(320) P21_DP2_DIFF_TRYKK &700  ; B2104 - B2103
AND>(320) B2215_PT &2000
RSET 222.05

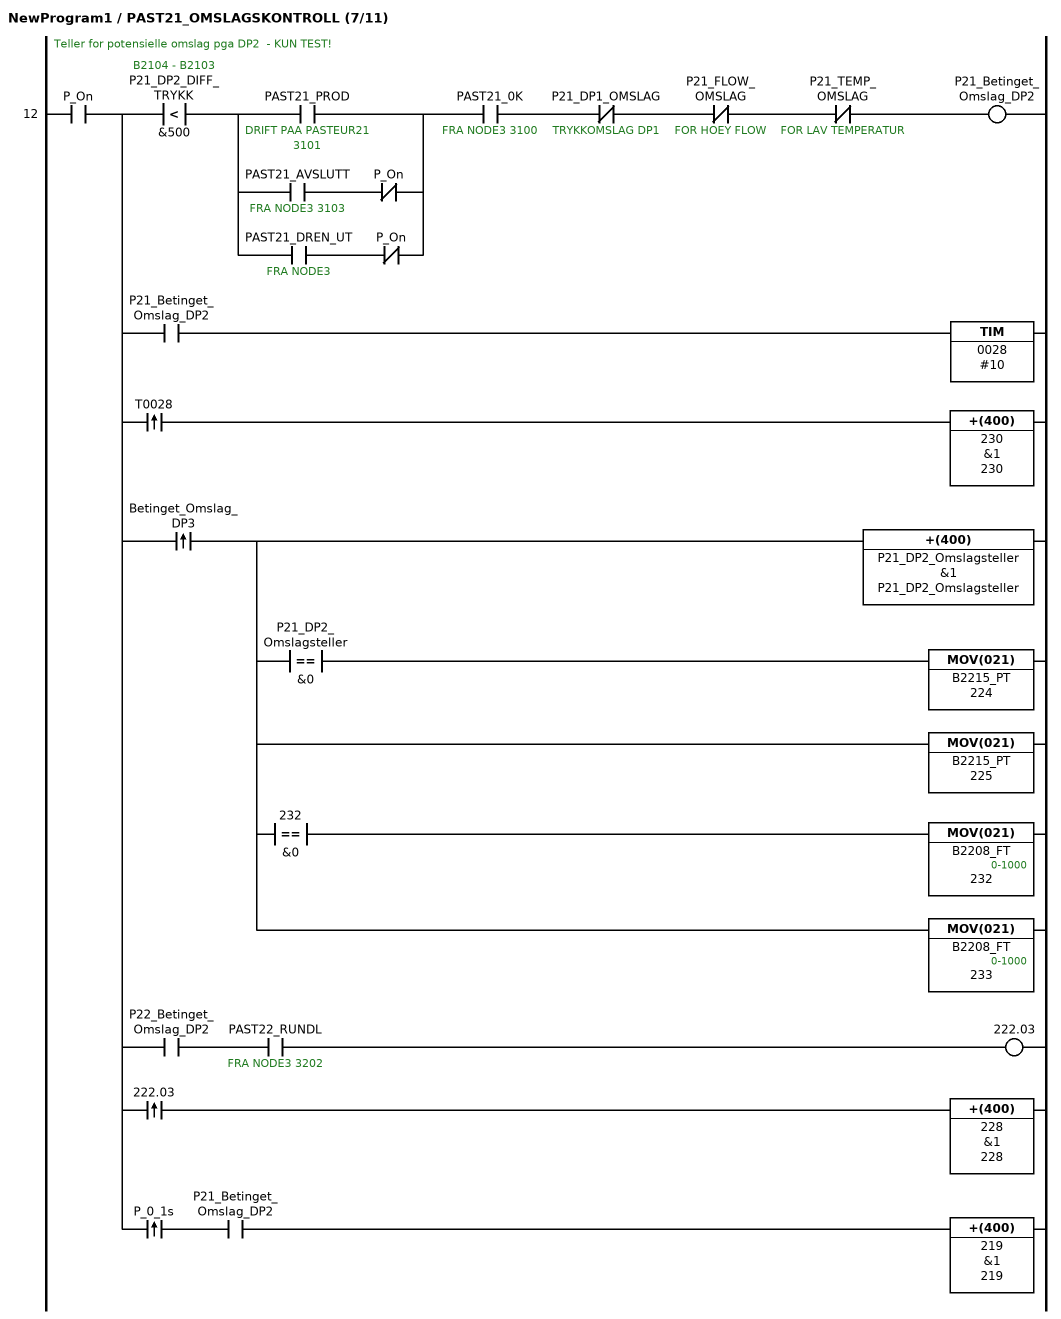
; rung 12: Teller for potensielle omslag pga DP2  - KUN TEST!
LD P_On
OUT TR0
AND<SL(313) P21_DP2_DIFF_TRYKK &500  ; B2104 - B2103
LD PAST21_PROD  ; DRIFT PAA PASTEUR21 3101
LD PAST21_AVSLUTT  ; FRA NODE3 3103
ANDNOT P_On
ORLD
LD PAST21_DREN_UT  ; FRA NODE3
ANDNOT P_On
ORLD
ANDLD
AND PAST21_0K  ; FRA NODE3 3100
ANDNOT P21_DP1_OMSLAG  ; TRYKKOMSLAG DP1
ANDNOT P21_FLOW_OMSLAG  ; FOR HOEY FLOW
ANDNOT P21_TEMP_OMSLAG  ; FOR LAV TEMPERATUR
OUT P21_Betinget_Omslag_DP2
LD TR0
AND P21_Betinget_Omslag_DP2
TIM 0028 #10
LD TR0
@AND T0028
+(400) 230 &1 230
LD TR0
@AND Betinget_Omslag_DP3
OUT TR1
+(400) P21_DP2_Omslagsteller &1 P21_DP2_Omslagsteller
AND=(300) P21_DP2_Omslagsteller &0
MOV(021) B2215_PT 224
LD TR1
MOV(021) B2215_PT 225
AND=(300) 232 &0
MOV(021) B2208_FT 232  ; 0-1000
LD TR1
MOV(021) B2208_FT 233  ; 0-1000
LD TR0
AND P22_Betinget_Omslag_DP2
AND PAST22_RUNDL  ; FRA NODE3 3202
OUT 222.03
LD TR0
@AND 222.03
+(400) 228 &1 228
LD TR0
@AND P_0_1s
AND P21_Betinget_Omslag_DP2
+(400) 219 &1 219

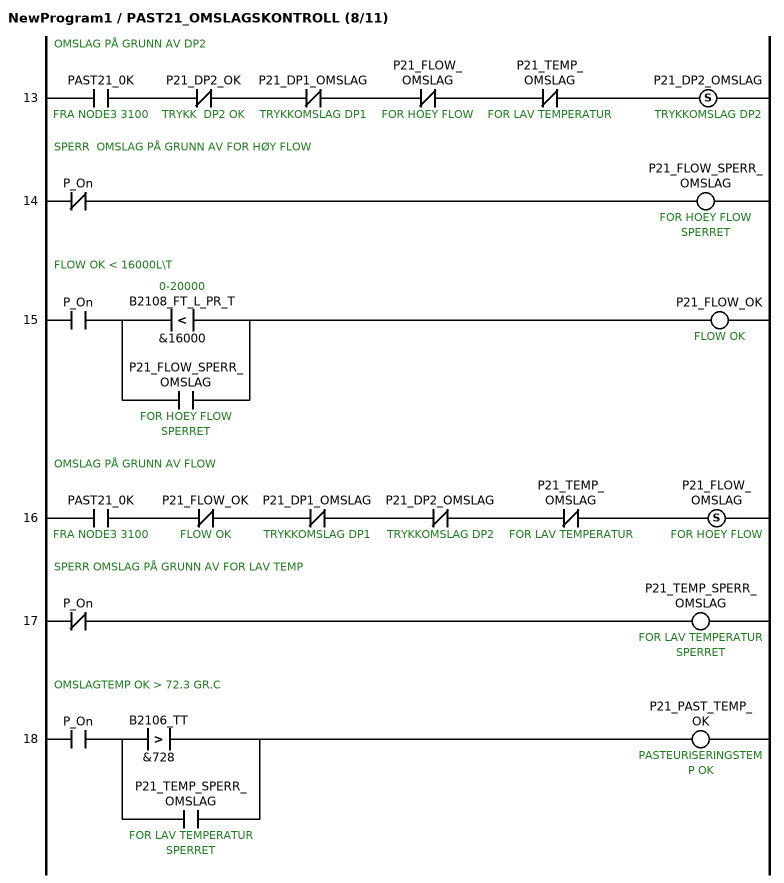
; rung 13: OMSLAG PÅ GRUNN AV DP2
LD PAST21_0K  ; FRA NODE3 3100
ANDNOT P21_DP2_OK  ; TRYKK  DP2 OK
ANDNOT P21_DP1_OMSLAG  ; TRYKKOMSLAG DP1
ANDNOT P21_FLOW_OMSLAG  ; FOR HOEY FLOW
ANDNOT P21_TEMP_OMSLAG  ; FOR LAV TEMPERATUR
SET P21_DP2_OMSLAG  ; TRYKKOMSLAG DP2
; rung 14: SPERR  OMSLAG PÅ GRUNN AV FOR HØY FLOW
LDNOT P_On  // CF113 INVERTERES OM SPERRING AV OMSLAG VED FOR HØY FLOW SKAL OPPHEVES
OUT P21_FLOW_SPERR_OMSLAG  ; FOR HOEY FLOW SPERRET
; rung 15: FLOW OK < 16000L\T
LD P_On
LD<(310) B2108_FT_L_PR_T &16000  ; 0-20000
OR P21_FLOW_SPERR_OMSLAG  ; FOR HOEY FLOW SPERRET
ANDLD
OUT P21_FLOW_OK  ; FLOW OK
; rung 16: OMSLAG PÅ GRUNN AV FLOW
LD PAST21_0K  ; FRA NODE3 3100
ANDNOT P21_FLOW_OK  ; FLOW OK
ANDNOT P21_DP1_OMSLAG  ; TRYKKOMSLAG DP1
ANDNOT P21_DP2_OMSLAG  ; TRYKKOMSLAG DP2
ANDNOT P21_TEMP_OMSLAG  ; FOR LAV TEMPERATUR
SET P21_FLOW_OMSLAG  ; FOR HOEY FLOW
; rung 17: SPERR OMSLAG PÅ GRUNN AV FOR LAV TEMP
LDNOT P_On  // CF113 INVERTERES OM SPERRING AV OMSLAG VED FOR LAV OMSLAGSTEMPERATUR
OUT P21_TEMP_SPERR_OMSLAG  ; FOR LAV TEMPERATUR SPERRET
; rung 18: OMSLAGTEMP OK > 72.3 GR.C
LD P_On
LD>(320) B2106_TT &728
OR P21_TEMP_SPERR_OMSLAG  ; FOR LAV TEMPERATUR SPERRET
ANDLD
OUT P21_PAST_TEMP_OK  ; PASTEURISERINGSTEMP OK

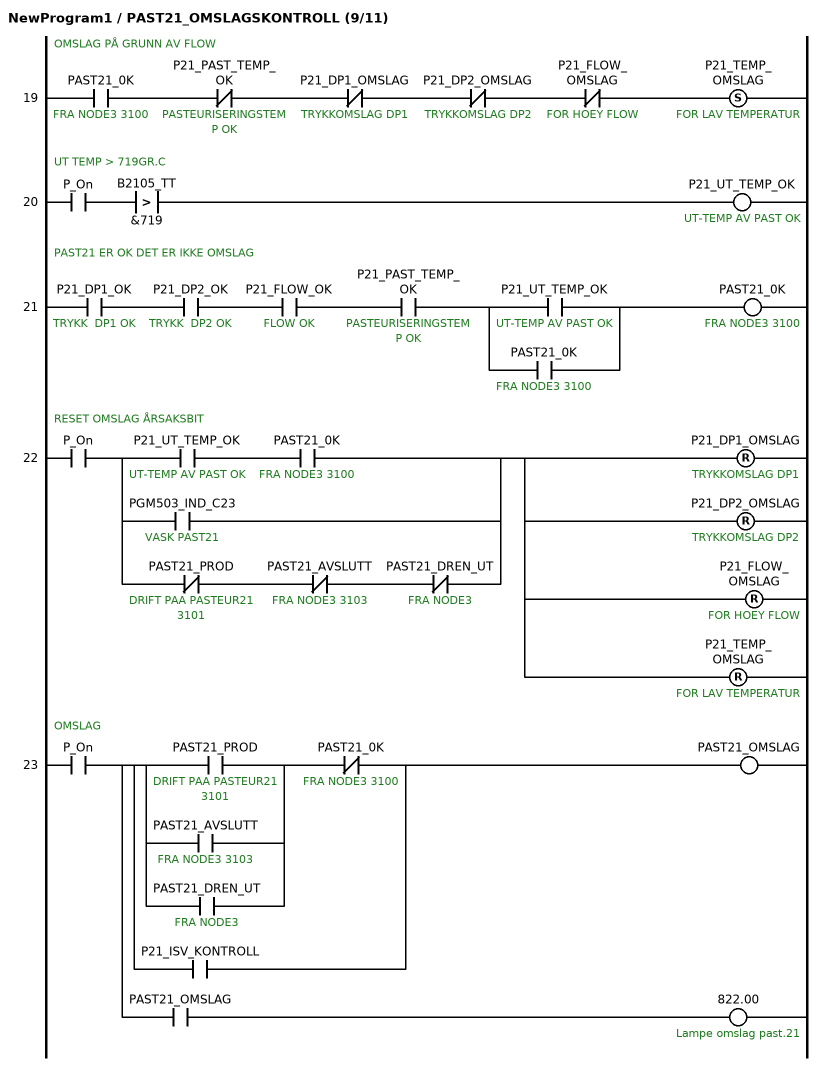
; rung 19: OMSLAG PÅ GRUNN AV FLOW
LD PAST21_0K  ; FRA NODE3 3100
ANDNOT P21_PAST_TEMP_OK  ; PASTEURISERINGSTEMP OK
ANDNOT P21_DP1_OMSLAG  ; TRYKKOMSLAG DP1
ANDNOT P21_DP2_OMSLAG  ; TRYKKOMSLAG DP2
ANDNOT P21_FLOW_OMSLAG  ; FOR HOEY FLOW
SET P21_TEMP_OMSLAG  ; FOR LAV TEMPERATUR
; rung 20: UT TEMP > 719GR.C
LD P_On
AND>(320) B2105_TT &719
OUT P21_UT_TEMP_OK  ; UT-TEMP AV PAST OK
; rung 21: PAST21 ER OK DET ER IKKE OMSLAG
LD P21_DP1_OK  ; TRYKK  DP1 OK
AND P21_DP2_OK  ; TRYKK  DP2 OK
AND P21_FLOW_OK  ; FLOW OK
AND P21_PAST_TEMP_OK  ; PASTEURISERINGSTEMP OK
LD P21_UT_TEMP_OK  ; UT-TEMP AV PAST OK
OR PAST21_0K  ; FRA NODE3 3100
ANDLD
OUT PAST21_0K  ; FRA NODE3 3100
; rung 22: RESET OMSLAG ÅRSAKSBIT
LD P_On
LD P21_UT_TEMP_OK  ; UT-TEMP AV PAST OK
AND PAST21_0K  ; FRA NODE3 3100
OR PGM503_IND_C23  ; VASK PAST21
LDNOT PAST21_PROD  ; DRIFT PAA PASTEUR21 3101
ANDNOT PAST21_AVSLUTT  ; FRA NODE3 3103
ANDNOT PAST21_DREN_UT  ; FRA NODE3
ORLD
ANDLD
RSET P21_DP1_OMSLAG  ; TRYKKOMSLAG DP1
RSET P21_DP2_OMSLAG  ; TRYKKOMSLAG DP2
RSET P21_FLOW_OMSLAG  ; FOR HOEY FLOW
RSET P21_TEMP_OMSLAG  ; FOR LAV TEMPERATUR
; rung 23: OMSLAG
LD P_On
OUT TR0
LD PAST21_PROD  ; DRIFT PAA PASTEUR21 3101
OR PAST21_AVSLUTT  ; FRA NODE3 3103
OR PAST21_DREN_UT  ; FRA NODE3
ANDNOT PAST21_0K  ; FRA NODE3 3100
OR P21_ISV_KONTROLL
ANDLD
OUT PAST21_OMSLAG
LD TR0
AND PAST21_OMSLAG
OUT 822.00  ; Lampe omslag past.21

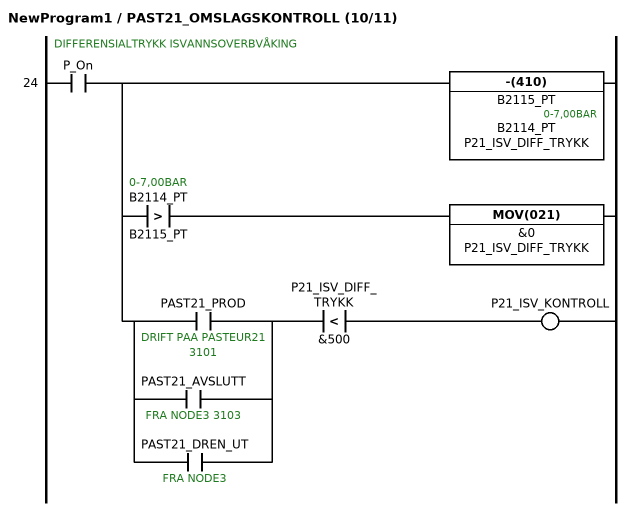
; rung 24: DIFFERENSIALTRYKK ISVANNSOVERBVÅKING
LD P_On
OUT TR0
-(410) B2115_PT B2114_PT P21_ISV_DIFF_TRYKK  ; 0-7,00BAR
AND>(320) B2114_PT B2115_PT  ; 0-7,00BAR
MOV(021) &0 P21_ISV_DIFF_TRYKK
LD TR0
LD PAST21_PROD  ; DRIFT PAA PASTEUR21 3101
OR PAST21_AVSLUTT  ; FRA NODE3 3103
OR PAST21_DREN_UT  ; FRA NODE3
ANDLD
AND<(310) P21_ISV_DIFF_TRYKK &500
OUT P21_ISV_KONTROLL

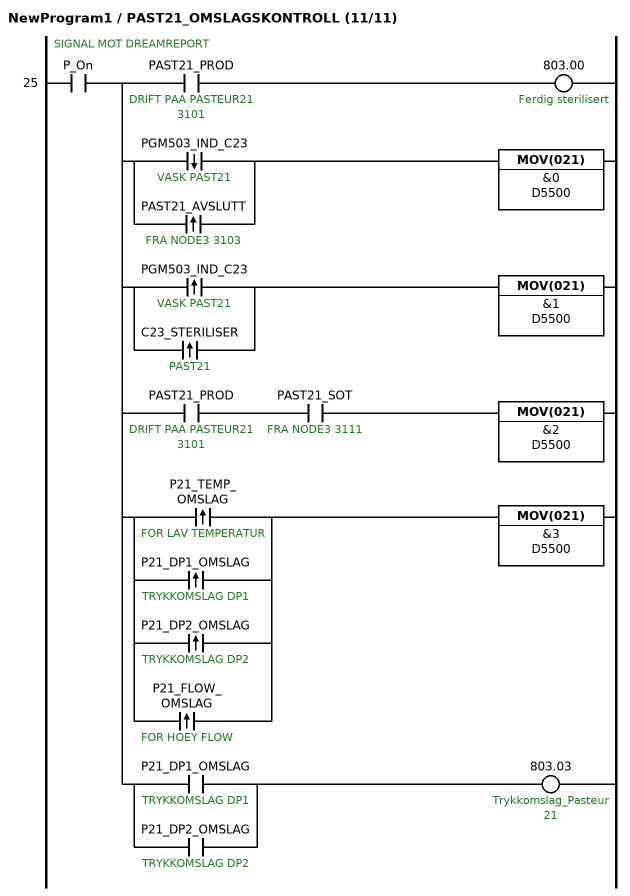
; rung 25: SIGNAL MOT DREAMREPORT
LD P_On
OUT TR0
AND PAST21_PROD  ; DRIFT PAA PASTEUR21 3101
OUT 803.00  ; Ferdig sterilisert
LD TR0
%LD PGM503_IND_C23  ; VASK PAST21
@OR PAST21_AVSLUTT  ; FRA NODE3 3103
ANDLD
MOV(021) &0 D5500
LD TR0
@LD PGM503_IND_C23  ; VASK PAST21
@OR C23_STERILISER  ; PAST21
ANDLD
MOV(021) &1 D5500
LD TR0
AND PAST21_PROD  ; DRIFT PAA PASTEUR21 3101
AND PAST21_SOT  ; FRA NODE3 3111
MOV(021) &2 D5500
LD TR0
@LD P21_TEMP_OMSLAG  ; FOR LAV TEMPERATUR
@OR P21_DP1_OMSLAG  ; TRYKKOMSLAG DP1
@OR P21_DP2_OMSLAG  ; TRYKKOMSLAG DP2
@OR P21_FLOW_OMSLAG  ; FOR HOEY FLOW
ANDLD
MOV(021) &3 D5500
LD TR0
LD P21_DP1_OMSLAG  ; TRYKKOMSLAG DP1
OR P21_DP2_OMSLAG  ; TRYKKOMSLAG DP2
ANDLD
OUT 803.03  ; Trykkomslag_Pasteur 21
; rung 26: Ingen_kommentar_funnet

### Section P2101_FLOWKONTROLL

